// TIA Portal project "LAB5" (V18)

(* hardware
DEVICE "S7-1500/ET200MP station_1"  S7-1500 station
   slot 0: "Rail_0"  Rack  6ES7 590-1***0-0AA0
   slot 1: "PLC_1"  CPU 1511-1 PN  6ES7 511-1AK00-0AB0  V1.0
      slot 3: "CPU display_1"  6ES7591-1XA00-0AA0
      slot 32768: "PROFINET interface_1"  X1
   slot 2: "CM 1542-5_1"  CM 1542-5  6GK7 542-5DX00-0XE0  V1.0
   slot 3: "DI 16x24VDC HF_1"  DI 16x24VDC HF  6ES7 521-1BH00-0AB0  V1.0
   slot 4: "DQ 16x24VDC/0.5A ST_1"  DQ 16x24VDC/0.5A ST  6ES7 522-1BH00-0AB0  V2.0
   slot 5: "AI 8xU/I/RTD/TC ST_1"  AI 8xU/I/RTD/TC ST  6ES7 531-7KF00-0AB0  V1.0
   slot 6: "AQ 4xU/I ST_1"  AQ 4xU/I ST  6ES7 532-5HD00-0AB0  V1.0
DEVICE "GSD device_1"  GSD.Device
   slot 0: "Rack_0"  Rail
   slot 0: "Slave_1"  6SE640X-1PB00-0AA0  V1.0
DEVICE "HMI_1"  KTP600 Basic color PN
   slot 0: "HMI_1"  KTP600 Basic color PN  6AV6 647-0AD11-3AX0  12.0.0.0
   slot 1: "HMI_RT_1"  KTP600 Basic color PN  6AV6 647-0AD11-3AX0  12.0.0.0
   slot 5: "HMI_1.IE_CP_1"  PROFINET Interface  12.0.0.0
      slot 1: "PROFINET Interface_1"  PROFINET Interface
         slot 1: "Port_1"  Port
DEVICE "PC-System_1"  SIMATIC PC station
   slot 0: "SIMATIC PC station"  Rail  SIMATIC PC-Station  V1.0
      slot 125: "Stationmanager"  Station_Manager  V6.0.4
   slot 1: "HMI_RT_2"  WinCC RT Advanced  6AV2 104-0xxxx-xxxx  16.0.0.0
      slot 33792: "Computer interface"  Host interface
   slot 2: "IE general_1"  IE General  IE_CP  V8.2.0
      slot 1: "PROFINET interface"  IEGeneral.Interface.8.2.0
*)

// ===== PLC "PLC_1"  CPU 1511-1 PN =====

VAR_GLOBAL   // PLC tag table "Default tag table"
   "Start_FIO" AT %I20.0 : Bool;
   "Stop_FIO" AT %I20.1 : Bool;
   "PE_FIO" AT %I20.2 : Bool;
   "Start_F" AT %I0.3 : Bool;
   "Stop_F" AT %I0.4 : Bool;
   "PE_F" AT %I0.5 : Bool;
   "Start_HMI" AT %M0.6 : Bool;
   "Stop_HMI" AT %M0.7 : Bool;
   "PE_HIM" AT %M1.0 : Bool;
   "I_LVL_SENSOR" AT %IW102 : Int;
   "Potenciometro" AT %IW100 : Int;
   "M_Start_Global" AT %M10.0 : Bool;
   "M_Stop_Global" AT %M10.1 : Bool;
   "M_PE_Global" AT %M10.2 : Bool;
   "LVL_CM" AT %MD20 : Real;
   "LVL_%" AT %MD24 : Real;
   "PV (Cm)" AT %MD30 : Real;
   "Tag_2" AT %MD340 : Real;
   "PV (%)" AT %MD34 : Real;
   "CV (%)" AT %MD36 : Real;
   "V_llenado" AT %QW100 : Int;
   "V_Descarga" AT %QW102 : Int;
   "LED_PID" AT %Q0.0 : Bool;
   "Start_Variador" AT %M0.0 : Bool;
   "VV_LLENADO" AT %M0.1 : Bool;
   "Tag_1" AT %M0.2 : Bool;
   "Tag_3" AT %M0.3 : Bool;
   "Tag_4" AT %M0.4 : Bool;
   "Tag_5" AT %M0.5 : Bool;
   "Tag_6" AT %M30.1 : Bool;
   "Tag_7" AT %M30.2 : Bool;
   "Tag_8" AT %M30.3 : Bool;
   "Tag_9" AT %M30.4 : Bool;
   "Tag_10" AT %M30.5 : Bool;
   "Tag_11" AT %M30.6 : Bool;
   "Tag_12" AT %M30.7 : Bool;
   "Tag_13" AT %M31.0 : Bool;
   "Tag_14" AT %M31.1 : Bool;
   "Tag_15" AT %M31.2 : Bool;
   "Tag_16" AT %M31.3 : Bool;
   "palabraestado" AT %IW26 : Word;
   "Palabramando" AT %QW18 : Word;
   "velocidadescribir" AT %QW20 : Int;
   "parametro" AT %QW10 : Word;
   "indice" AT %QW12 : Word;
   "valorparametro" AT %QD14 : DWord;
   "leerparametro" AT %IW18 : Word;
   "paramrecib" AT %MW4 : Word;
   "leerindice" AT %IW20 : Word;
   "indicerecib" AT %MW6 : Word;
   "leervalparametro" AT %ID22 : DWord;
   "valorparamrecib" AT %MD8 : DWord;
   "GREEN" AT %Q0.1 : Bool;
   "SP_ALCANZADO" AT %M40.0 : Bool;
   "AMARILLO" AT %Q0.2 : Bool;
   "RED" AT %Q0.3 : Bool;
   "Sel_Factory" AT %I20.3 : Bool;
   "Sel_HMI_BD_WCC" AT %I20.4 : Bool;
   "SETP_%" AT %MD100 : Real;
   "SP_HMI" AT %MD60 : Real;
   "SP_DB" AT %MD64 : Real;
   "SP_DBN" AT %MD70 : Real;
   "SP_WCC" AT %MW74 : Int;
   "lvl_cm(1)" AT %QW104 : Word;
   "PV_FIO" AT %QW106 : Word;
   "PE_WinCC" AT %M50.0 : Bool;
   "Stop_WinCC" AT %M50.1 : Bool;
   "Start_WinCC" AT %M50.2 : Bool;
   "Nivel_Maximo" AT %M50.3 : Bool;
   "Nivel_Minimo" AT %M50.4 : Bool;
   "SEL_WCC" AT %I20.5 : Bool;
END_VAR

TYPE "inn"
   STRUCT
      Mandoderecha : Bool;
      Mandoizquierdo : Bool;
      ControldesdePLC : Bool;
      Inversionvalorconsigna : Bool;
      Noutilizado : Bool;
      Potenciometrohaciaarriba : Bool;
      Potenciometrohaciaabajo : Bool;
      "Local/remoto" : Bool;
      "ON/OFF1" : Bool;
      OFF2stopelectrico : Bool;
      OFF3stoprapido : Bool;
      Activarpulsos : Bool;
      Activargeneradorrampa : Bool;
      Generadorrampa : Bool;
      Activarvalorconsigna : Bool;
      Acusedefallo : Bool;
      Velocidadvariador : Int;
   END_STRUCT;
END_TYPE

TYPE "out"
   STRUCT
      Sindesviacionvalreaconsigna : Bool;
      Controlsolicitado : Bool;
      frecuenciasalida : Bool;
      alarma : Bool;
      freno : Bool;
      sobrecarga : Bool;
      giro : Bool;
      sobrecargaconvertidor : Bool;
      listoparaservicio : Bool;
      listoparaarrancar : Bool;
      serviciodesbloqueado : Bool;
      fallo : Bool;
      "comando aus2/off2" : Bool;
      "comandoaus3/off3" : Bool;
      Bloqueodearranque : Bool;
      Alarmas : Bool;
      Velocidadactual : Int;
   END_STRUCT;
END_TYPE

DATA_BLOCK "Red_variador"   // DB1
{ S7_Optimized_Access := 'FALSE' }
VERSION : 0.1
   VAR
      estadovariador : "out";
   END_VAR
BEGIN
END_DATA_BLOCK

DATA_BLOCK "Señal Sensor_DB"   // DB2
{ S7_Optimized_Access := 'TRUE' }
VERSION : 0.1
// stored: InstanceOfName Señal Sensor
"Señal Sensor"
BEGIN
END_DATA_BLOCK

DATA_BLOCK "Salida PID_DB"   // DB3
{ S7_Optimized_Access := 'TRUE' }
VERSION : 0.1
// stored: InstanceOfName Salida PID
"Salida PID"
BEGIN
END_DATA_BLOCK

DATA_BLOCK "Alarmas_DB_1"   // DB5
{ S7_Optimized_Access := 'TRUE' }
VERSION : 0.1
// stored: InstanceOfName Alarmas
"Alarmas"
BEGIN
END_DATA_BLOCK

DATA_BLOCK "Variador_1_DB"   // DB6
{ S7_Optimized_Access := 'TRUE' }
VERSION : 0.1
// stored: InstanceOfName Variador_1
"Variador_1"
BEGIN
END_DATA_BLOCK

DATA_BLOCK "Selector_DB"   // DB7
{ S7_Optimized_Access := 'TRUE' }
VERSION : 0.1
// stored: InstanceOfName Selector
"Selector"
BEGIN
END_DATA_BLOCK

DATA_BLOCK "Selector_DB_1"   // DB8
{ S7_Optimized_Access := 'TRUE' }
VERSION : 0.1
// stored: InstanceOfName Selector
"Selector"
BEGIN
END_DATA_BLOCK

DATA_BLOCK "Alarmas_DB"   // DB9
{ S7_Optimized_Access := 'TRUE' }
VERSION : 0.1
// stored: InstanceOfName Alarmas
"Alarmas"
BEGIN
END_DATA_BLOCK

DATA_BLOCK "SetPointCM_DB"   // DB10
{ S7_Optimized_Access := 'TRUE' }
VERSION : 0.1
// stored: InstanceOfName SetPointCM
"SetPointCM"
BEGIN
END_DATA_BLOCK

DATA_BLOCK "scada_variador"   // DB11
{ S7_Optimized_Access := 'FALSE' }
VERSION : 0.1
   VAR
      esc_variador : "inn";
   END_VAR
BEGIN
END_DATA_BLOCK

DATA_BLOCK "Selector_DB_2"   // DB12
{ S7_Optimized_Access := 'TRUE' }
VERSION : 0.1
// stored: InstanceOfName Selector
"Selector"
BEGIN
END_DATA_BLOCK

DATA_BLOCK "Selector_DB_3"   // DB13
{ S7_Optimized_Access := 'TRUE' }
VERSION : 0.1
// stored: InstanceOfName Selector
"Selector"
BEGIN
END_DATA_BLOCK

DATA_BLOCK "ON/OFF_DB"   // DB14
{ S7_Optimized_Access := 'TRUE' }
VERSION : 0.1
// stored: InstanceOfName ON/OFF
"ON/OFF"
BEGIN
END_DATA_BLOCK

DATA_BLOCK "ON/OFF_DB_1"   // DB15
{ S7_Optimized_Access := 'TRUE' }
VERSION : 0.1
// stored: InstanceOfName ON/OFF
"ON/OFF"
BEGIN
END_DATA_BLOCK

DATA_BLOCK "Selector_DB_4"   // DB16
{ S7_Optimized_Access := 'TRUE' }
VERSION : 0.1
// stored: InstanceOfName Selector
"Selector"
BEGIN
END_DATA_BLOCK

FUNCTION_BLOCK "SetPointCM"   // FB1, LAD
{ S7_Optimized_Access := 'TRUE' }
VERSION : 0.1
   VAR_INPUT
      InAnalog : Int;
      NivelMAX : Real;
   END_VAR
   VAR_OUTPUT
      "Nivel (Cm)." : Real;
      "Nivel (%)" : Real;
   END_VAR
   VAR
      Aux : Real;
   END_VAR
BEGIN

REGION Network 1
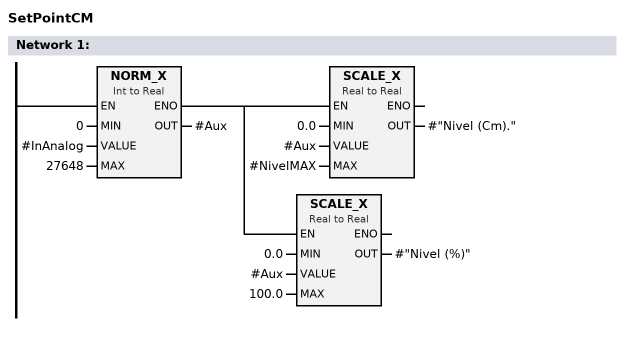
   RUNG wire#powerrail
      { S7_Templates := "[SrcType := Int, DestType := Real]" } Normalize(min := 0, value := #InAnalog, max := 27648, out => #Aux)
      wire#w1
      { S7_Templates := "[SrcType := Real, DestType := Real]" } Scale(min := 0.0, value := #Aux, max := #NivelMAX, out => #"Nivel (Cm).")
   END_RUNG
   RUNG wire#w1
      { S7_Templates := "[SrcType := Real, DestType := Real]" } Scale(min := 0.0, value := #Aux, max := 100.0, out => #"Nivel (%)")
   END_RUNG
   // the same network as SCL:
   #Aux := NORM_X(MIN := 0, VALUE := #InAnalog, MAX := 27648);
   #"Nivel (Cm)." := SCALE_X(MIN := 0.0, VALUE := #Aux, MAX := #NivelMAX);
   #"Nivel (%)" := SCALE_X(MIN := 0.0, VALUE := #Aux, MAX := 100.0);
END_REGION
END_FUNCTION_BLOCK

FUNCTION_BLOCK "Señal Sensor"   // FB2, LAD
{ S7_Optimized_Access := 'TRUE' }
VERSION : 0.1
   VAR_INPUT
      InAnalog : Int;
      NivelMax : Real;
   END_VAR
   VAR_OUTPUT
      "Nivel (Cm)" : Real;
      "Nivel (%)" : Real;
   END_VAR
   VAR
      Aux : Real;
   END_VAR
BEGIN

REGION Network 1
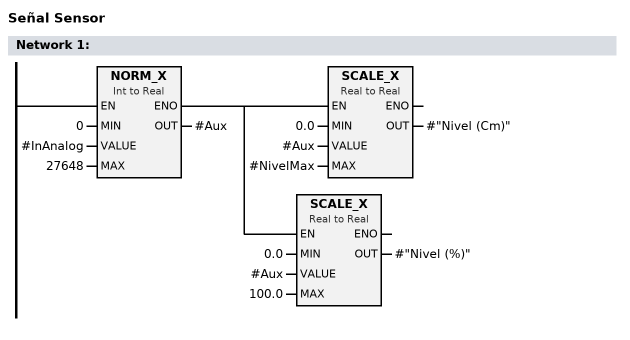
   RUNG wire#powerrail
      { S7_Templates := "[SrcType := Int, DestType := Real]" } Normalize(min := 0, value := #InAnalog, max := 27648, out => #Aux)
      wire#w1
      { S7_Templates := "[SrcType := Real, DestType := Real]" } Scale(min := 0.0, value := #Aux, max := #NivelMax, out => #"Nivel (Cm)")
   END_RUNG
   RUNG wire#w1
      { S7_Templates := "[SrcType := Real, DestType := Real]" } Scale(min := 0.0, value := #Aux, max := 100.0, out => #"Nivel (%)")
   END_RUNG
   // the same network as SCL:
   #Aux := NORM_X(MIN := 0, VALUE := #InAnalog, MAX := 27648);
   #"Nivel (Cm)" := SCALE_X(MIN := 0.0, VALUE := #Aux, MAX := #NivelMax);
   #"Nivel (%)" := SCALE_X(MIN := 0.0, VALUE := #Aux, MAX := 100.0);
END_REGION
END_FUNCTION_BLOCK

FUNCTION_BLOCK "Salida PID"   // FB3, LAD
{ S7_Optimized_Access := 'TRUE' }
VERSION : 0.1
   VAR_INPUT
      SalidaPID : Real;
   END_VAR
   VAR_OUTPUT
      V_llenado : Int;
      V_Descarga : Int;
   END_VAR
   VAR
      SalidaPID_Aux : Real;
      Aux : Real;
      OutAnlog : Int;
   END_VAR
BEGIN

REGION Network 1
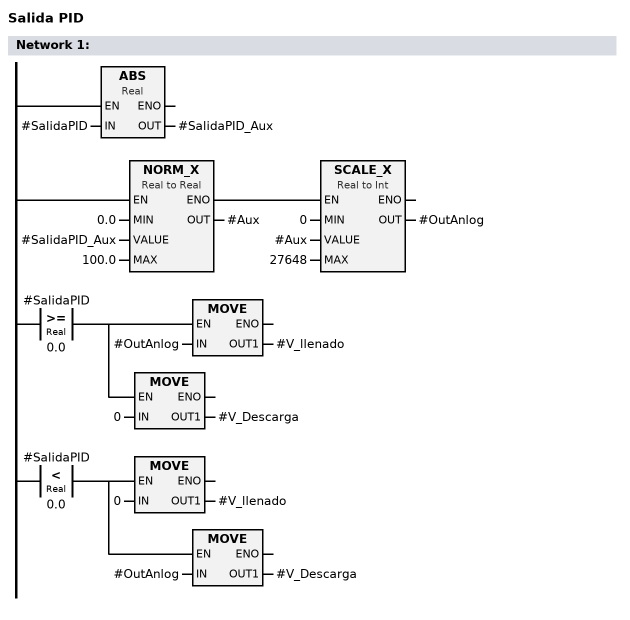
   RUNG wire#powerrail
      { S7_Templates := "SrcType := Real" } Abs(in := #SalidaPID, out => #SalidaPID_Aux)
   END_RUNG
   RUNG wire#powerrail
      { S7_Templates := "[SrcType := Real, DestType := Real]" } Normalize(min := 0.0, value := #SalidaPID_Aux, max := 100.0, out => #Aux)
      { S7_Templates := "[SrcType := Real, DestType := Int]" } Scale(min := 0, value := #Aux, max := 27648, out => #OutAnlog)
   END_RUNG
   RUNG wire#powerrail
      { S7_Templates := "SrcType := Real" } GE_Contact(in1 := #SalidaPID, in2 := 0.0)
      wire#w1
      Move(in := #OutAnlog, out1 => #V_llenado)
   END_RUNG
   RUNG wire#w1
      Move(in := 0, out1 => #V_Descarga)
   END_RUNG
   RUNG wire#powerrail
      { S7_Templates := "SrcType := Real" } LT_Contact(in1 := #SalidaPID, in2 := 0.0)
      wire#w2
      Move(in := 0, out1 => #V_llenado)
   END_RUNG
   RUNG wire#w2
      Move(in := #OutAnlog, out1 => #V_Descarga)
   END_RUNG
   // the same network as SCL:
   #SalidaPID_Aux := ABS(#SalidaPID);
   #Aux := NORM_X(MIN := 0.0, VALUE := #SalidaPID_Aux, MAX := 100.0);
   #OutAnlog := SCALE_X(MIN := 0, VALUE := #Aux, MAX := 27648);
   IF #SalidaPID >= 0.0 THEN
       #V_llenado := #OutAnlog;
       #V_Descarga := 0;
   END_IF;
   IF #SalidaPID < 0.0 THEN
       #V_llenado := 0;
       #V_Descarga := #OutAnlog;
   END_IF;
END_REGION
END_FUNCTION_BLOCK

FUNCTION_BLOCK "Alarmas"   // FB4, LAD
{ S7_Optimized_Access := 'TRUE' }
VERSION : 0.1
   VAR_INPUT
      Sistema_Activo : Bool;
      SP_Alcanzado : Bool;
   END_VAR
   VAR_OUTPUT
      Q_Luz_Run : Bool;
      Q_Alarma_SP : Bool;
   END_VAR
   VAR
      Timer_Pulse_1 : IEC_TIMER;
      Timer_Pulse_2 : IEC_TIMER;
      Timer_2Seg : IEC_TIMER;
      Aux_Flag_SP : Bool;
   END_VAR
BEGIN

REGION Network 1
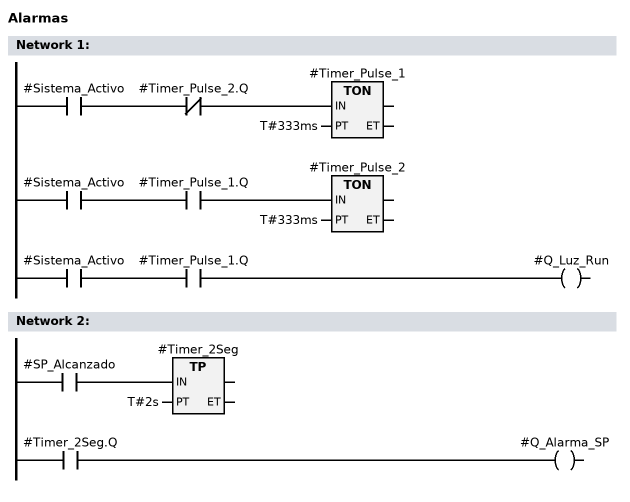
   #Timer_Pulse_1.TON(IN := #Sistema_Activo AND NOT #Timer_Pulse_2.Q, PT := T#333ms);
   #Timer_Pulse_2.TON(IN := #Sistema_Activo AND #Timer_Pulse_1.Q, PT := T#333ms);
   #Q_Luz_Run := #Sistema_Activo AND #Timer_Pulse_1.Q;
END_REGION

REGION Network 2
   #Timer_2Seg.TP(IN := #SP_Alcanzado, PT := T#2s);
   #Q_Alarma_SP := #Timer_2Seg.Q;
END_REGION
END_FUNCTION_BLOCK

FUNCTION_BLOCK "Variador_1"   // FB5, LAD
{ S7_Optimized_Access := 'TRUE' }
VERSION : 0.1
BEGIN

REGION Network 1
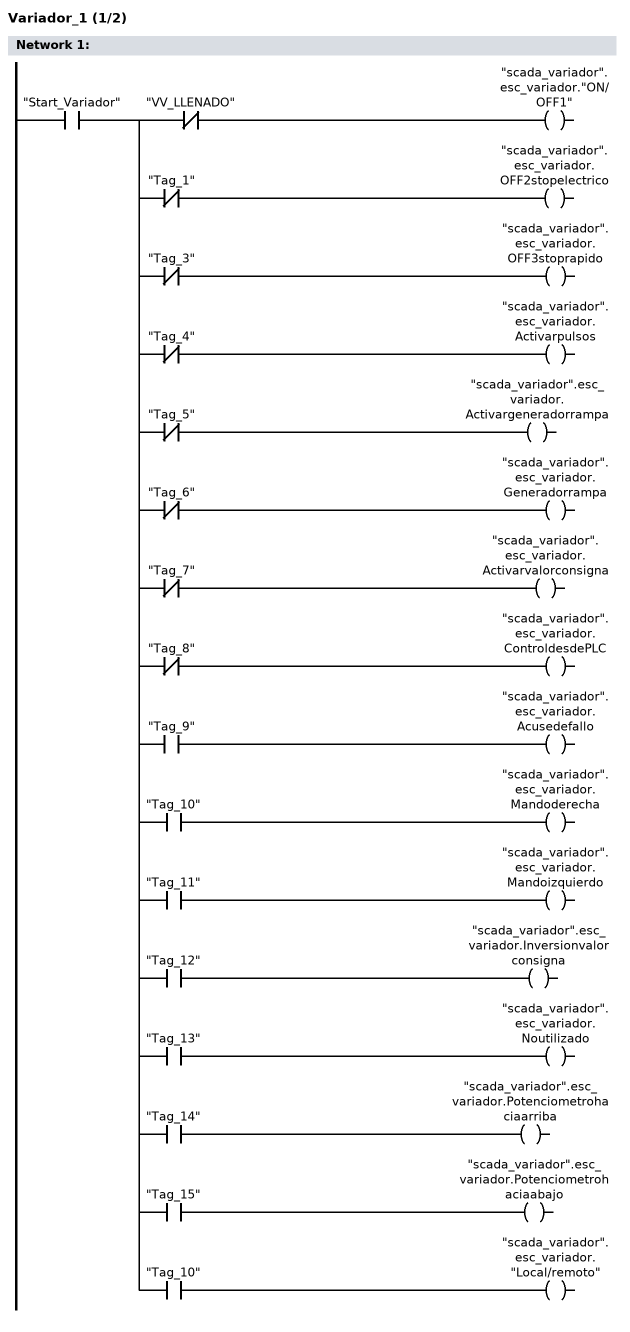
   RUNG wire#powerrail
      Contact( "Start_Variador" )
      wire#w1
      I_Contact( "VV_LLENADO" )
      Coil( "scada_variador".esc_variador."ON/OFF1" )
   END_RUNG
   RUNG wire#w1
      I_Contact( "Tag_1" )
      Coil( "scada_variador".esc_variador.OFF2stopelectrico )
   END_RUNG
   RUNG wire#w1
      I_Contact( "Tag_3" )
      Coil( "scada_variador".esc_variador.OFF3stoprapido )
   END_RUNG
   RUNG wire#w1
      I_Contact( "Tag_4" )
      Coil( "scada_variador".esc_variador.Activarpulsos )
   END_RUNG
   RUNG wire#w1
      I_Contact( "Tag_5" )
      Coil( "scada_variador".esc_variador.Activargeneradorrampa )
   END_RUNG
   RUNG wire#w1
      I_Contact( "Tag_6" )
      Coil( "scada_variador".esc_variador.Generadorrampa )
   END_RUNG
   RUNG wire#w1
      I_Contact( "Tag_7" )
      Coil( "scada_variador".esc_variador.Activarvalorconsigna )
   END_RUNG
   RUNG wire#w1
      I_Contact( "Tag_8" )
      Coil( "scada_variador".esc_variador.ControldesdePLC )
   END_RUNG
   RUNG wire#w1
      Contact( "Tag_9" )
      Coil( "scada_variador".esc_variador.Acusedefallo )
   END_RUNG
   RUNG wire#w1
      Contact( "Tag_10" )
      Coil( "scada_variador".esc_variador.Mandoderecha )
   END_RUNG
   RUNG wire#w1
      Contact( "Tag_11" )
      Coil( "scada_variador".esc_variador.Mandoizquierdo )
   END_RUNG
   RUNG wire#w1
      Contact( "Tag_12" )
      Coil( "scada_variador".esc_variador.Inversionvalorconsigna )
   END_RUNG
   RUNG wire#w1
      Contact( "Tag_13" )
      Coil( "scada_variador".esc_variador.Noutilizado )
   END_RUNG
   RUNG wire#w1
      Contact( "Tag_14" )
      Coil( "scada_variador".esc_variador.Potenciometrohaciaarriba )
   END_RUNG
   RUNG wire#w1
      Contact( "Tag_15" )
      Coil( "scada_variador".esc_variador.Potenciometrohaciaabajo )
   END_RUNG
   RUNG wire#w1
      Contact( "Tag_10" )
      Coil( "scada_variador".esc_variador."Local/remoto" )
   END_RUNG
   // the same network as SCL:
   "scada_variador".esc_variador."ON/OFF1" := "Start_Variador" AND NOT "VV_LLENADO";
   "scada_variador".esc_variador.OFF2stopelectrico := "Start_Variador" AND NOT "Tag_1";
   "scada_variador".esc_variador.OFF3stoprapido := "Start_Variador" AND NOT "Tag_3";
   "scada_variador".esc_variador.Activarpulsos := "Start_Variador" AND NOT "Tag_4";
   "scada_variador".esc_variador.Activargeneradorrampa := "Start_Variador" AND NOT "Tag_5";
   "scada_variador".esc_variador.Generadorrampa := "Start_Variador" AND NOT "Tag_6";
   "scada_variador".esc_variador.Activarvalorconsigna := "Start_Variador" AND NOT "Tag_7";
   "scada_variador".esc_variador.ControldesdePLC := "Start_Variador" AND NOT "Tag_8";
   "scada_variador".esc_variador.Acusedefallo := "Start_Variador" AND "Tag_9";
   "scada_variador".esc_variador.Mandoderecha := "Start_Variador" AND "Tag_10";
   "scada_variador".esc_variador.Mandoizquierdo := "Start_Variador" AND "Tag_11";
   "scada_variador".esc_variador.Inversionvalorconsigna := "Start_Variador" AND "Tag_12";
   "scada_variador".esc_variador.Noutilizado := "Start_Variador" AND "Tag_13";
   "scada_variador".esc_variador.Potenciometrohaciaarriba := "Start_Variador" AND "Tag_14";
   "scada_variador".esc_variador.Potenciometrohaciaabajo := "Start_Variador" AND "Tag_15";
   "scada_variador".esc_variador."Local/remoto" := "Start_Variador" AND "Tag_10";
END_REGION

REGION Network 2
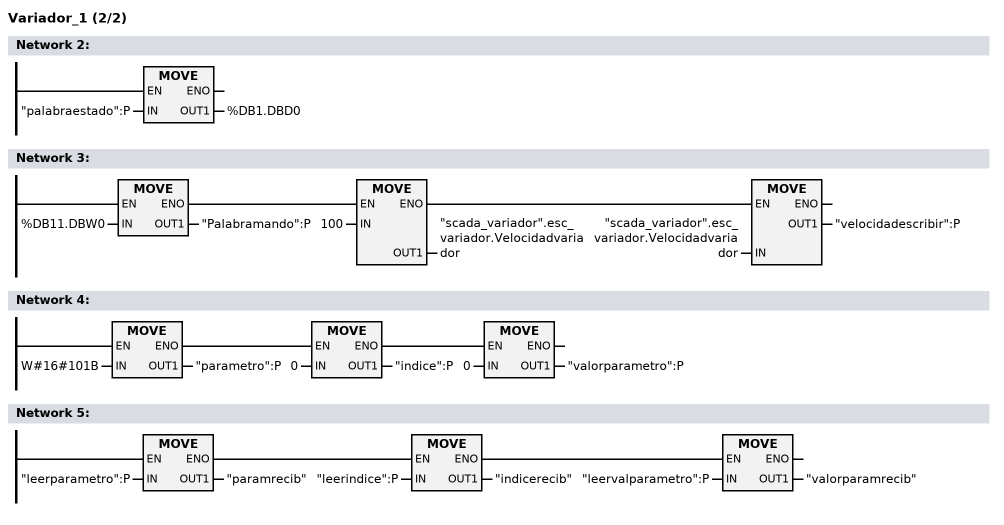
   RUNG wire#powerrail
      Move(in := "palabraestado":P, out1 => %DB1.DBD0)
   END_RUNG
   // the same network as SCL:
   %DB1.DBD0 := "palabraestado":P;
END_REGION

REGION Network 3
   RUNG wire#powerrail
      Move(in := %DB11.DBW0, out1 => "Palabramando":P)
      Move(in := 100, out1 => "scada_variador".esc_variador.Velocidadvariador)
      Move(in := "scada_variador".esc_variador.Velocidadvariador, out1 => "velocidadescribir":P)
   END_RUNG
   // the same network as SCL:
   "Palabramando":P := %DB11.DBW0;
   "scada_variador".esc_variador.Velocidadvariador := 100;
   "velocidadescribir":P := "scada_variador".esc_variador.Velocidadvariador;
END_REGION

REGION Network 4
   RUNG wire#powerrail
      Move(in := W#16#101B, out1 => "parametro":P)
      Move(in := 0, out1 => "indice":P)
      Move(in := 0, out1 => "valorparametro":P)
   END_RUNG
   // the same network as SCL:
   "parametro":P := W#16#101B;
   "indice":P := 0;
   "valorparametro":P := 0;
END_REGION

REGION Network 5
   RUNG wire#powerrail
      Move(in := "leerparametro":P, out1 => "paramrecib")
      Move(in := "leerindice":P, out1 => "indicerecib")
      Move(in := "leervalparametro":P, out1 => "valorparamrecib")
   END_RUNG
   // the same network as SCL:
   "paramrecib" := "leerparametro":P;
   "indicerecib" := "leerindice":P;
   "valorparamrecib" := "leervalparametro":P;
END_REGION
END_FUNCTION_BLOCK

FUNCTION_BLOCK "Selector"   // FB6, LAD
{ S7_Optimized_Access := 'TRUE' }
VERSION : 0.1
   VAR_INPUT
      Pot_Factory_In : Real;
      SetPoint_HMI_In : Real;
      SetPoint_DB_In : Real;
      SetPoint_WCC_In : Real;
      SetPoint_DBN_In : Real;
      PosSel_1 : Bool;
      PosSel_2 : Bool;
      PosSel_3 : Bool;
   END_VAR
   VAR_OUTPUT
      Setpoint_Final : Real;
   END_VAR
   VAR
      SEL_1 : Bool;
      SEL_2 : Bool;
      Sel_V1 : Bool;
      Sel_v2 : Bool;
   END_VAR
BEGIN

REGION Network 1
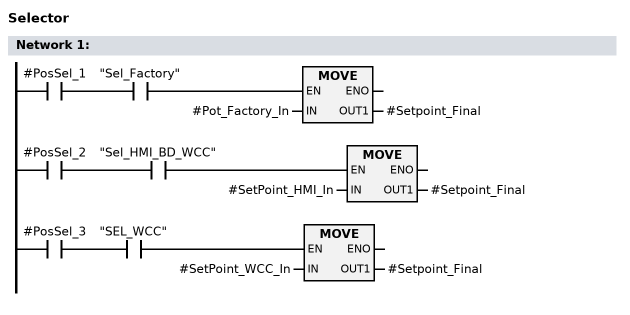
   RUNG wire#powerrail
      Contact( #PosSel_1 )
      Contact( "Sel_Factory" )
      Move(in := #Pot_Factory_In, out1 => #Setpoint_Final)
   END_RUNG
   RUNG wire#powerrail
      Contact( #PosSel_2 )
      Contact( "Sel_HMI_BD_WCC" )
      Move(in := #SetPoint_HMI_In, out1 => #Setpoint_Final)
   END_RUNG
   RUNG wire#powerrail
      Contact( #PosSel_3 )
      Contact( "SEL_WCC" )
      Move(in := #SetPoint_WCC_In, out1 => #Setpoint_Final)
   END_RUNG
   // the same network as SCL:
   IF #PosSel_1 AND "Sel_Factory" THEN #Setpoint_Final := #Pot_Factory_In; END_IF;
   IF #PosSel_2 AND "Sel_HMI_BD_WCC" THEN #Setpoint_Final := #SetPoint_HMI_In; END_IF;
   IF #PosSel_3 AND "SEL_WCC" THEN #Setpoint_Final := #SetPoint_WCC_In; END_IF;
END_REGION
END_FUNCTION_BLOCK

FUNCTION_BLOCK "ON/OFF"   // FB7, LAD
{ S7_Optimized_Access := 'TRUE' }
VERSION : 0.1
   VAR_INPUT
      "SP_ON/OFF" : Real;
      Sensor : Real;
   END_VAR
   VAR_OUTPUT
      P1 : Int;
      P2 : Int;
   END_VAR
   VAR
      Aux1 : Real;
      Aux2 : Real;
      OutAnlog : Int;
   END_VAR
   VAR_TEMP   // added for the SCL form of the ladder/FBD networks
      _w1 : Bool;
      _w2 : Bool;
   END_VAR
BEGIN

REGION Network 1
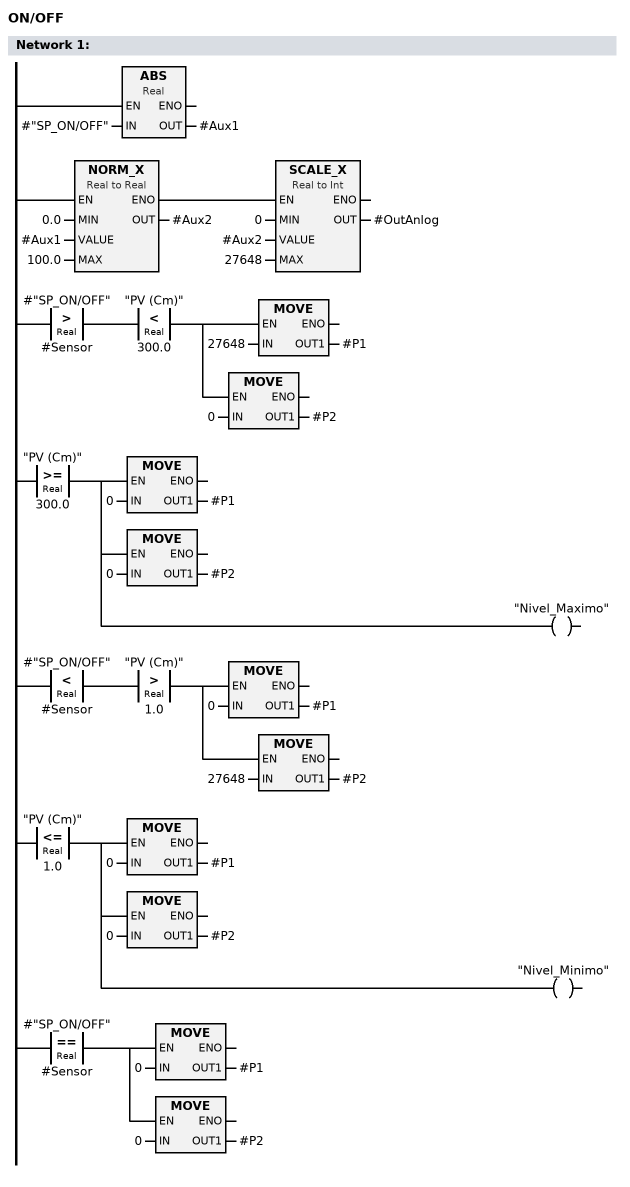
   RUNG wire#powerrail
      { S7_Templates := "SrcType := Real" } Abs(in := #"SP_ON/OFF", out => #Aux1)
   END_RUNG
   RUNG wire#powerrail
      { S7_Templates := "[SrcType := Real, DestType := Real]" } Normalize(min := 0.0, value := #Aux1, max := 100.0, out => #Aux2)
      { S7_Templates := "[SrcType := Real, DestType := Int]" } Scale(min := 0, value := #Aux2, max := 27648, out => #OutAnlog)
   END_RUNG
   RUNG wire#powerrail
      { S7_Templates := "SrcType := Real" } GT_Contact(in1 := #"SP_ON/OFF", in2 := #Sensor)
      { S7_Templates := "SrcType := Real" } LT_Contact(in1 := "PV (Cm)", in2 := 300.0)
      wire#w1
      Move(in := 27648, out1 => #P1)
   END_RUNG
   RUNG wire#w1
      Move(in := 0, out1 => #P2)
   END_RUNG
   RUNG wire#powerrail
      { S7_Templates := "SrcType := Real" } GE_Contact(in1 := "PV (Cm)", in2 := 300.0)
      wire#w2
      Move(in := 0, out1 => #P1)
   END_RUNG
   RUNG wire#w2
      Move(in := 0, out1 => #P2)
   END_RUNG
   RUNG wire#w2
      Coil( "Nivel_Maximo" )
   END_RUNG
   RUNG wire#powerrail
      { S7_Templates := "SrcType := Real" } LT_Contact(in1 := #"SP_ON/OFF", in2 := #Sensor)
      { S7_Templates := "SrcType := Real" } GT_Contact(in1 := "PV (Cm)", in2 := 1.0)
      wire#w3
      Move(in := 0, out1 => #P1)
   END_RUNG
   RUNG wire#w3
      Move(in := 27648, out1 => #P2)
   END_RUNG
   RUNG wire#powerrail
      { S7_Templates := "SrcType := Real" } LE_Contact(in1 := "PV (Cm)", in2 := 1.0)
      wire#w4
      Move(in := 0, out1 => #P1)
   END_RUNG
   RUNG wire#w4
      Move(in := 0, out1 => #P2)
   END_RUNG
   RUNG wire#w4
      Coil( "Nivel_Minimo" )
   END_RUNG
   RUNG wire#powerrail
      { S7_Templates := "SrcType := Real" } EQ_Contact(in1 := #"SP_ON/OFF", in2 := #Sensor)
      wire#w5
      Move(in := 0, out1 => #P1)
   END_RUNG
   RUNG wire#w5
      Move(in := 0, out1 => #P2)
   END_RUNG
   // the same network as SCL:
   #Aux1 := ABS(#"SP_ON/OFF");
   #Aux2 := NORM_X(MIN := 0.0, VALUE := #Aux1, MAX := 100.0);
   #OutAnlog := SCALE_X(MIN := 0, VALUE := #Aux2, MAX := 27648);
   IF (#"SP_ON/OFF" > #Sensor) AND ("PV (Cm)" < 300.0) THEN
       #P1 := 27648;
       #P2 := 0;
   END_IF;
   #_w1 := "PV (Cm)" >= 300.0;
   IF #_w1 THEN
       #P1 := 0;
       #P2 := 0;
   END_IF;
   "Nivel_Maximo" := #_w1;
   IF (#"SP_ON/OFF" < #Sensor) AND ("PV (Cm)" > 1.0) THEN
       #P1 := 0;
       #P2 := 27648;
   END_IF;
   #_w2 := "PV (Cm)" <= 1.0;
   IF #_w2 THEN
       #P1 := 0;
       #P2 := 0;
   END_IF;
   "Nivel_Minimo" := #_w2;
   IF #"SP_ON/OFF" = #Sensor THEN
       #P1 := 0;
       #P2 := 0;
   END_IF;
END_REGION
END_FUNCTION_BLOCK

ORGANIZATION_BLOCK "Main"   // OB1, LAD, ProgramCycle
TITLE = "Main Program Sweep (Cycle)"
{ S7_Optimized_Access := 'TRUE' }
VERSION : 0.1
   VAR_INPUT
      Initial_Call : Bool;   // Initial call of this OB
      Remanence : Bool;   // =True, if remanent data are available
   END_VAR
   VAR_TEMP
      l : Bool;
      l1 : DWord;
   END_VAR
BEGIN

REGION Network 1
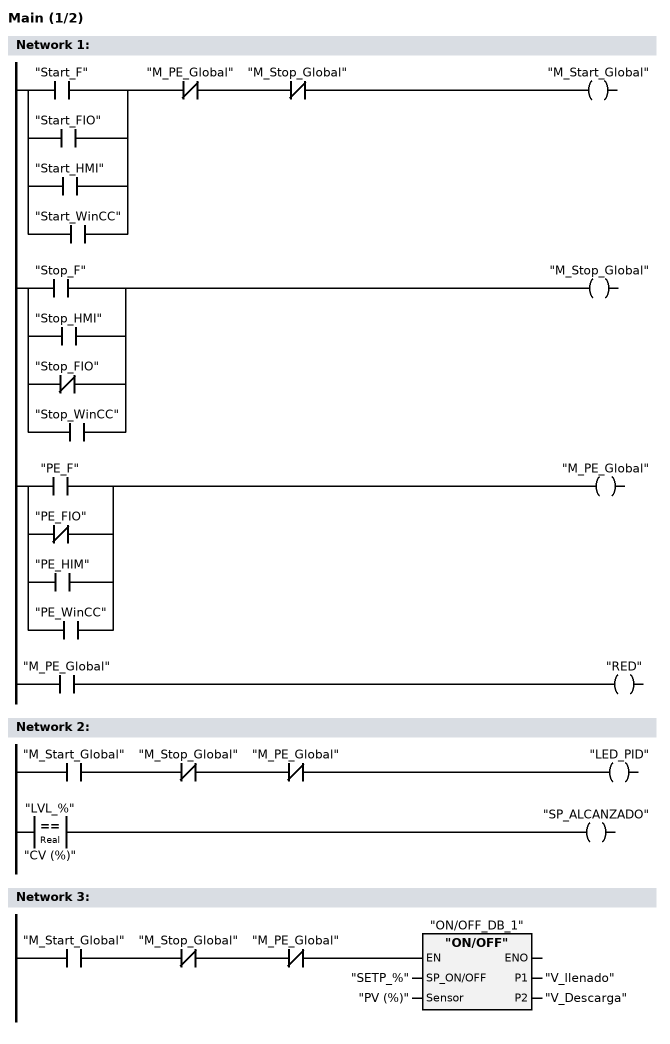
   RUNG wire#powerrail
      Contact( "Start_F" )
      wire#w1
      I_Contact( "M_PE_Global" )
      I_Contact( "M_Stop_Global" )
      Coil( "M_Start_Global" )
   END_RUNG
   RUNG wire#powerrail
      Contact( "Start_FIO" )
   END_RUNG wire#w1
   RUNG wire#powerrail
      Contact( "Start_HMI" )
   END_RUNG wire#w1
   RUNG wire#powerrail
      Contact( "Start_WinCC" )
   END_RUNG wire#w1
   RUNG wire#powerrail
      Contact( "Stop_F" )
      wire#w2
      Coil( "M_Stop_Global" )
   END_RUNG
   RUNG wire#powerrail
      Contact( "Stop_HMI" )
   END_RUNG wire#w2
   RUNG wire#powerrail
      I_Contact( "Stop_FIO" )
   END_RUNG wire#w2
   RUNG wire#powerrail
      Contact( "Stop_WinCC" )
   END_RUNG wire#w2
   RUNG wire#powerrail
      Contact( "PE_F" )
      wire#w3
      Coil( "M_PE_Global" )
   END_RUNG
   RUNG wire#powerrail
      I_Contact( "PE_FIO" )
   END_RUNG wire#w3
   RUNG wire#powerrail
      Contact( "PE_HIM" )
   END_RUNG wire#w3
   RUNG wire#powerrail
      Contact( "PE_WinCC" )
   END_RUNG wire#w3
   RUNG wire#powerrail
      Contact( "M_PE_Global" )
      Coil( "RED" )
   END_RUNG
   // the same network as SCL:
   "M_Start_Global" := ("Start_F" OR "Start_FIO" OR "Start_HMI" OR "Start_WinCC") AND NOT "M_PE_Global" AND NOT "M_Stop_Global";
   "M_Stop_Global" := "Stop_F" OR "Stop_HMI" OR NOT "Stop_FIO" OR "Stop_WinCC";
   "M_PE_Global" := "PE_F" OR NOT "PE_FIO" OR "PE_HIM" OR "PE_WinCC";
   "RED" := "M_PE_Global";
END_REGION

REGION Network 2
   RUNG wire#powerrail
      Contact( "M_Start_Global" )
      I_Contact( "M_Stop_Global" )
      I_Contact( "M_PE_Global" )
      Coil( "LED_PID" )
   END_RUNG
   RUNG wire#powerrail
      { S7_Templates := "SrcType := Real" } EQ_Contact(in1 := "LVL_%", in2 := "CV (%)")
      Coil( "SP_ALCANZADO" )
   END_RUNG
   // the same network as SCL:
   "LED_PID" := "M_Start_Global" AND NOT "M_Stop_Global" AND NOT "M_PE_Global";
   "SP_ALCANZADO" := "LVL_%" = "CV (%)";
END_REGION

REGION Network 3
   RUNG wire#powerrail
      Contact( "M_Start_Global" )
      I_Contact( "M_Stop_Global" )
      I_Contact( "M_PE_Global" )
      "ON/OFF_DB_1"("SP_ON/OFF" := "SETP_%", Sensor := "PV (%)", P1 => "V_llenado", P2 => "V_Descarga")
   END_RUNG
   // the same network as SCL:
   IF "M_Start_Global" AND NOT "M_Stop_Global" AND NOT "M_PE_Global" THEN
       "ON/OFF_DB_1"("SP_ON/OFF" := "SETP_%", Sensor := "PV (%)", P1 => "V_llenado", P2 => "V_Descarga");   // "ON/OFF"
   END_IF;
END_REGION

REGION Network 4
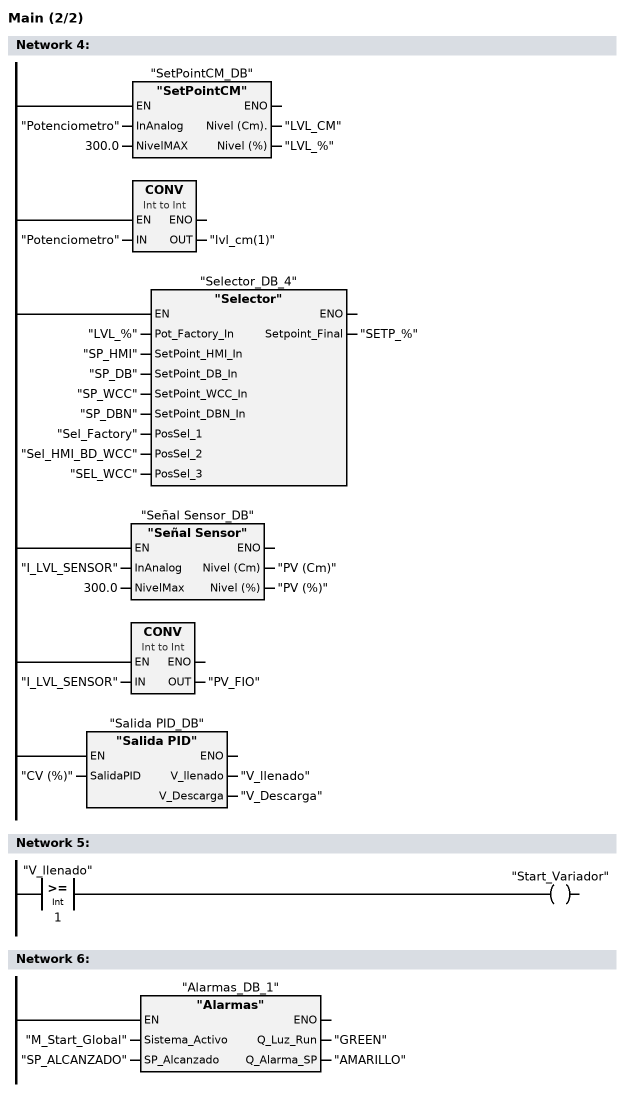
   RUNG wire#powerrail
      "SetPointCM_DB"(InAnalog := "Potenciometro", NivelMAX := 300.0, "Nivel (Cm)." => "LVL_CM", "Nivel (%)" => "LVL_%")
   END_RUNG
   RUNG wire#powerrail
      { S7_Templates := "[SrcType := Int, DestType := Int]" } Convert(in := "Potenciometro", out => "lvl_cm(1)")
   END_RUNG
   RUNG wire#powerrail
      "Selector_DB_4"(Pot_Factory_In := "LVL_%", SetPoint_HMI_In := "SP_HMI", SetPoint_DB_In := "SP_DB", SetPoint_WCC_In := "SP_WCC", SetPoint_DBN_In := "SP_DBN", PosSel_1 := "Sel_Factory", PosSel_2 := "Sel_HMI_BD_WCC", PosSel_3 := "SEL_WCC", Setpoint_Final => "SETP_%")
   END_RUNG
   RUNG wire#powerrail
      "Señal Sensor_DB"(InAnalog := "I_LVL_SENSOR", NivelMax := 300.0, "Nivel (Cm)" => "PV (Cm)", "Nivel (%)" => "PV (%)")
   END_RUNG
   RUNG wire#powerrail
      { S7_Templates := "[SrcType := Int, DestType := Int]" } Convert(in := "I_LVL_SENSOR", out => "PV_FIO")
   END_RUNG
   RUNG wire#powerrail
      "Salida PID_DB"(SalidaPID := "CV (%)", V_llenado => "V_llenado", V_Descarga => "V_Descarga")
   END_RUNG
   // the same network as SCL:
   "SetPointCM_DB"(InAnalog := "Potenciometro",   // "SetPointCM"
                   NivelMAX := 300.0,
                   "Nivel (Cm)." => "LVL_CM",
                   "Nivel (%)" => "LVL_%");
   "lvl_cm(1)" := INT_TO_INT("Potenciometro");
   "Selector_DB_4"(Pot_Factory_In := "LVL_%",   // "Selector"
                   SetPoint_HMI_In := "SP_HMI",
                   SetPoint_DB_In := "SP_DB",
                   SetPoint_WCC_In := "SP_WCC",
                   SetPoint_DBN_In := "SP_DBN",
                   PosSel_1 := "Sel_Factory",
                   PosSel_2 := "Sel_HMI_BD_WCC",
                   PosSel_3 := "SEL_WCC",
                   Setpoint_Final => "SETP_%");
   "Señal Sensor_DB"(InAnalog := "I_LVL_SENSOR",   // "Señal Sensor"
                     NivelMax := 300.0,
                     "Nivel (Cm)" => "PV (Cm)",
                     "Nivel (%)" => "PV (%)");
   "PV_FIO" := INT_TO_INT("I_LVL_SENSOR");
   "Salida PID_DB"(SalidaPID := "CV (%)", V_llenado => "V_llenado", V_Descarga => "V_Descarga");   // "Salida PID"
END_REGION

REGION Network 5
   RUNG wire#powerrail
      { S7_Templates := "SrcType := Int" } GE_Contact(in1 := "V_llenado", in2 := 1)
      Coil( "Start_Variador" )
   END_RUNG
   // the same network as SCL:
   "Start_Variador" := "V_llenado" >= 1;
END_REGION

REGION Network 6
   RUNG wire#powerrail
      "Alarmas_DB_1"(Sistema_Activo := "M_Start_Global", SP_Alcanzado := "SP_ALCANZADO", Q_Luz_Run => "GREEN", Q_Alarma_SP => "AMARILLO")
   END_RUNG
   // the same network as SCL:
   "Alarmas_DB_1"(Sistema_Activo := "M_Start_Global",   // "Alarmas"
                  SP_Alcanzado := "SP_ALCANZADO",
                  Q_Luz_Run => "GREEN",
                  Q_Alarma_SP => "AMARILLO");
END_REGION
END_ORGANIZATION_BLOCK

ORGANIZATION_BLOCK "PIDA"   // OB30, LAD, CyclicInterrupt
{ S7_Optimized_Access := 'TRUE' }
VERSION : 0.1
   VAR_INPUT
      Initial_Call : Bool;   // Initial call of this OB
      Event_Count : Int;   // Events discarded
   END_VAR
BEGIN

REGION Network 1
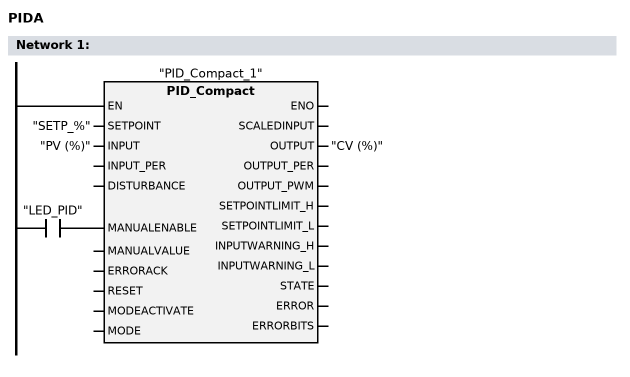
   "PID_Compact_1"(Setpoint := "SETP_%", Input := "PV (%)", ManualEnable := "LED_PID", Output => "CV (%)");   // PID_Compact
END_REGION
END_ORGANIZATION_BLOCK

(* ===== HMI "HMI_RT_1" =====
system functions are stored by id; their names below are inferred from use
connection "HMI_Connection_3": ETHERNET, SMART_S7_1500_OMS

HMI tags "Default tag table"
   "Stop_HMI" : Bool = PLC Stop_HMI AT %M0.7, 1 s
   "Start_HMI" : Bool = PLC Start_HMI AT %M0.6, 1 s
   "M_Start_Global" : Bool = PLC M_Start_Global AT %M10.0, 1 s
   "M_Stop_Global" : Bool = PLC M_Stop_Global AT %M10.1, 1 s
   "M_PE_Global" : Bool = PLC M_PE_Global AT %M10.2, 1 s
   "CV (%)" : Real = PLC "CV (%)" AT %MD36, 1 s
   "LVL_CM" : Real = PLC LVL_CM AT %MD20, 1 s
   "LVL_%" : Real = PLC LVL_% AT %MD24, 1 s
   "GREEN" : Bool = PLC GREEN AT %Q0.1, 1 s
   "AMARILLO" : Bool = PLC AMARILLO AT %Q0.2, 1 s
   "RED" : Bool = PLC RED AT %Q0.3, 1 s
   "PE_HIM" : Bool = PLC PE_HIM AT %M1.0, 1 s
   "lvl_cm(1)" : Word = PLC "lvl_cm(1)" AT %QW104, 1 s
   "Nivel_Maximo" : Bool = PLC Nivel_Maximo AT %M50.3, 1 s
   "Nivel_Minimo" : Bool = PLC Nivel_Minimo AT %M50.4, 1 s
   "PV (%)" : Real = PLC "PV (%)" AT %MD34, 1 s
   "PV (Cm)" : Real = PLC "PV (Cm)" AT %MD30, 1 s
   "SP_HMI" : Real = PLC SP_HMI AT %MD60, 1 s
   "SETP_%" : Real = PLC SETP_% AT %MD100, 1 s

screen "Root screen" 320x240, template "Template_2"
   GraphicView "Graphic view_4" at 27,0 size 155x164; Picture "Graphic_4"
   Button "Button_2" at 124,207 size 62x27; TextOff 'Stop'
      on Press: InvertBit("Stop_HMI")
      Appearance <- "M_Stop_Global"
   Switch "Pushbutton_Emergency" at 0,196 size 47x44; CaptionText 'Switch'; TextOff '0'; TextOn '1'; PictureOff "Pushbutton_Emergency_Off_256c"; PictureOn "Pushbutton_Emergency_On_256c"
      on Change: InvertBit("M_PE_Global")
      ProcessValue <- "PE_HIM"
   Bar "Bar_1" at 46,36 size 120x98; MinimumValue 0; MaximumValue 300
      ProcessValue <- "PV (Cm)"
   GraphicView "Graphic view_5" at 0,0 size 28x84; Picture "Graphic_5"
   Button "Button_3" at 231,41 size 59x21; TextOff '100'
      on Press: SetTag("LVL_%", 100); SetTag("SP_HMI", 100)
   IOField "I/O field_1" at 238,157 size 77x21; FormatPattern s99999
      ProcessValue <- "SETP_%"
   TrendView "Trend view_1" at 350,109 size 203x197
   TextField "Text field_1" at 224,5 size 69x32; Text 'Referencia Rápida'
   Button "Button_4" at 231,62 size 59x19; TextOff '80'
      on Press: SetTag("LVL_%", 80); SetTag("SP_HMI", 80)
   Button "Button_5" at 231,81 size 59x19; TextOff '60'
      on Press: SetTag("LVL_%", 60); SetTag("SP_HMI", 60)
   Button "Button_6" at 231,100 size 59x15; TextOff '40'
      on Press: SetTag("LVL_%", 40); SetTag("SP_HMI", 40)
   Button "Button_7" at 231,114 size 59x17; TextOff '20'
      on Press: SetTag("LVL_%", 20); SetTag("SP_HMI", 20)
   Button "Button_8" at 231,131 size 59x14; TextOff '0'
      on Press: SetTag("LVL_%", 0); SetTag("SP_HMI", 0)
   Button "Button_9" at 250,208 size 68x30; TextOff 'Grafica'
      on Click: ActivateScreen("Screen_1", 0)
   Button "Button_1" at 58,207 size 53x27; TextOff 'star'
      on Press: InvertBit("Start_HMI")
      Appearance <- "M_Start_Global"
   Rectangle "Rectangle_1" at 0,3 size 23x14
      Appearance <- "GREEN"
   Rectangle "Rectangle_2" at 0,19 size 23x13
      Appearance <- "AMARILLO"
   Rectangle "Rectangle_3" at 0,34 size 23x13
      Appearance <- "RED"
   Circle "Circle_1" at 187,34 size 10x10
      Appearance <- "Nivel_Maximo"
   Circle "Circle_2" at 188,136 size 9x9
      Appearance <- "Nivel_Minimo"
   TextField "Text field_2" at 6,175 size 65x13; Text 'Nivel Actual:'
   TextField "Text field_3" at 180,158 size 59x13; Text 'Referencia:'
   IOField "I/O field_2" at 70,172 size 77x21; FormatPattern s99999
      ProcessValue <- "PV (%)"

Template "Template_1" 320x240
   Button "Exit" at 714,429 size 71x50; TextOn 'Exit'; TextOff 'Exit'; PictureOn "ExitRuntime_KTP700_Basic_PN_TR"; PictureOff "ExitRuntime_KTP700_Basic_PN_TR"
      on Release: StopRuntime(0)
   Button "Template_Button" at 614,429 size 71x50; TextOff 'Text'
   Button "Template_Button_1" at 514,429 size 71x50; TextOff 'Text'
   Button "Template_Button_2" at 414,429 size 71x50; TextOff 'Text'
   Button "Template_Button_3" at 314,429 size 71x50; TextOff 'Text'
   Button "Template_Button_4" at 214,429 size 71x50; TextOff 'Text'
   Button "Alarms" at 114,429 size 71x50; TextOn 'Alarms'; TextOff 'Alarms'; PictureOn "AlarmDisplay_KTP700_Basic_PN_TR"; PictureOff "AlarmDisplay_KTP700_Basic_PN_TR"
      on Release: function_ef3f5d25("Alarm window_Unacknowledged", -1)
   Button "Start screen" at 14,429 size 71x50; TextOn 'Start screen'; TextOff 'Start screen'; PictureOn "NavigateHome_KTP700_Basic_PN_TR"; PictureOff "NavigateHome_KTP700_Basic_PN_TR"
      on Release: ActivateScreen("Root screen", 0)
   DateTimeField "HmiScreenItemData" at 695,25 size 105x25
   DateTimeField "HmiScreenItemData_1" at 695,0 size 105x25
   GraphicView "Logo" at 0,0 size 91x51; Picture "Logo of HMI_1"

screen "Screen_1" 320x240
   TrendView "Trend view_1" at 30,54 size 258x174
   Button "Button_1" at 105,13 size 96x32; TextOff 'Volver'
      on Click: ActivateScreen("Root screen", 0)
*)

(* ===== HMI "HMI_RT_2" =====
system functions are stored by id; their names below are inferred from use
connection "HMI_Connection_2": ETHERNET, S7_1500_OMS

HMI tags "Default tag table"
   "Inicio1" : Bool = PLC Start_FIO AT %I20.0, 1 s
   "Sto1" : Bool = PLC Stop_FIO AT %I20.1, 1 s
   "M_Stop_Global" : Bool = PLC M_Stop_Global AT %M10.1, 1 s
   "M_Start_Global" : Bool = PLC M_Start_Global AT %M10.0, 1 s
   "Stop_WinCC" : Bool = PLC Stop_WinCC AT %M50.1, 1 s
   "Start_WinCC" : Bool = PLC Start_WinCC AT %M50.2, 1 s
   "PE_WinCC" : Bool = PLC PE_WinCC AT %M50.0, 1 s
   "GREEN" : Bool = PLC GREEN AT %Q0.1, 1 s
   "AMARILLO" : Bool = PLC AMARILLO AT %Q0.2, 1 s
   "RED" : Bool = PLC RED AT %Q0.3, 1 s
   "LVL_%" : Real = PLC LVL_% AT %MD24, 1 s
   "CV (%)" : Real = PLC "CV (%)" AT %MD36, 1 s
   "PV (Cm)" : Real = PLC "PV (Cm)" AT %MD30, 1 s
   "LVL_CM" : Real = PLC LVL_CM AT %MD20, 1 s
   "PV (%)" : Real = PLC "PV (%)" AT %MD34, 1 s
   "SETP_%" : Real = PLC SETP_% AT %MD100, 1 s
   "SP_WCC" : Int = PLC SP_WCC AT %MW74, 1 s
   "M_PE_Global" : Bool = PLC M_PE_Global AT %M10.2, 1 s

screen "Screen_1" 1024x768
   GraphicView "Graphic view_6" at 204,415 size 83x50; Picture "Graphic_12"
   GraphicView "Graphic view_4" at 150,218 size 187x217; Picture "Graphic_4"
   Switch "Pushbutton_Emergency" at 26,148 size 97x96; CaptionText 'Switch'; TextOff '0'; TextOn '1'; PictureOff "Pushbutton_Emergency_Off_256c"; PictureOn "Pushbutton_Emergency_On_256c"
      ObjectEnable <- "PE_WinCC"
      ProcessValue <- "PE_WinCC"
      on SwitchOn: SetTag("PE_WinCC", 1)
      on SwitchOff: SetTag("PE_WinCC", 0)
      Appearance <- "M_PE_Global"
   Bar "Bar_1" at 185,249 size 118x152; MinimumValue 0; MaximumValue 100
      ProcessValue <- "PV (%)"
   GraphicView "Graphic view_5" at 327,263 size 21x69; Picture "Graphic_5"
   TrendView "Trend view_1" at 478,70 size 505x331
   TextField "Text field_1" at 588,575 size 141x64; Text 'Referencia'
   TextField "Text field_3" at 220,15 size 543x40; Text 'Guía 5 Supervisión Filocaris, Andrés'
   TextField "Text field_6" at 13,243 size 125x18; Text 'Paro de Emergencia'
   Rectangle "Rectangle_1" at 326,266 size 21x14
      Appearance <- "GREEN"
   Rectangle "Rectangle_2" at 326,281 size 21x14
      Appearance <- "AMARILLO"
   Rectangle "Rectangle_3" at 326,296 size 21x14
      Appearance <- "RED"
   GraphicView "Graphic view_2" at 162,459 size 101x99; Picture "Graphic_10"
   GraphicView "Graphic view_3" at 207,149 size 75x75; Picture "Graphic_11"
   GraphicView "Graphic view_1" at 275,91 size 191x137; Picture "Graphic_15"
   Slider "Slider_1" at 304,617 size 689x80; Caption 'SIMATIC'
      ProcessValue <- "SP_WCC"
   Button "Button_1" at 27,38 size 96x32; TextOff 'Start'
      on Press: InvertBit("Start_WinCC")
      Appearance <- "M_Start_Global"
   Button "Button_2" at 27,87 size 96x32; TextOff 'Stop'
      on Press: InvertBit("Stop_WinCC")
      Appearance <- "M_Stop_Global"
*)